// TIA Portal project "kanalAlarmowySygDzwiek" (V15)

(* hardware
DEVICE "S7-1200 station_1"  S7-1200 Station
   slot 0: "Rack_0"  S7-1200 Rack  Rack  V1.0
   slot 1: "PLC_1"  CPU 1214C DC/DC/DC  6ES7 214-1AG40-0XB0  V4.2
      slot 3: "AQ 1x12BIT_1"  AQ1 signal board  6ES7 232-4HA30-0XB0  V1.0
   slot 101: "CM 1243-5"  CM 1243-5  6GK7 243-5DX30-0XE0  V1.3
   slot 102: "CM 1241 (RS485)_1"  CM 1241 (RS485)  6ES7 241-1CH30-0XB0  V1.0
DEVICE "S7-1200 station_2"  S7-1200 Station
   slot 0: "Rack_0"  S7-1200 Rack  Rack  V1.0
   slot 1: "PLC_2"  CPU 1212C DC/DC/DC  6ES7 212-1AE40-0XB0  V4.2
   slot 2: "AI 4x13BIT/AQ 2x14BIT_1"  6ES7 234-4HE32-0XB0  V2.0
*)

// ===== PLC "PLC_1"  CPU 1214C DC/DC/DC =====

VAR_GLOBAL   // PLC tag table "Default tag table"
   "Clock_Byte" AT %MB50 : Byte;
   "Clock_10Hz" AT %M50.0 : Bool;
   "Clock_5Hz" AT %M50.1 : Bool;
   "Clock_2.5Hz" AT %M50.2 : Bool;
   "Clock_2Hz" AT %M50.3 : Bool;
   "Clock_1.25Hz" AT %M50.4 : Bool;
   "Clock_1Hz" AT %M50.5 : Bool;
   "Clock_0.625Hz" AT %M50.6 : Bool;
   "Clock_0.5Hz" AT %M50.7 : Bool;
   "System_Byte" AT %MB1 : Byte;
   "FirstScan" AT %M1.0 : Bool;
   "DiagStatusUpdate" AT %M1.1 : Bool;
   "AlwaysTRUE" AT %M1.2 : Bool;
   "AlwaysFALSE" AT %M1.3 : Bool;
   "zaklocenie" AT %I0.0 : Bool;
   "potwierdzenie" AT %I0.7 : Bool;
   "Tag_1" AT %M10.0 : Bool;
   "Tag_2" AT %M10.1 : Bool;
   "sygnalizacja" AT %Q0.1 : Bool;
   "System_Byte(1)" AT %MB1 : Byte;
   "Tag_3" AT %I0.1 : Bool;
   "Tag_4" AT %I0.6 : Bool;
   "Tag_5" AT %M20.0 : Bool;
   "Tag_6" AT %Q0.2 : Bool;
   "czasTrwania" AT %MD30 : Time;
   "Tag_7" AT %M22.0 : Bool;
   "Tag_8" AT %M22.1 : Bool;
   "Tag_9" AT %M22.2 : Bool;
   "Tag_10" AT %M22.3 : Bool;
   "Tag_11" AT %Q0.3 : Bool;
   "Tag_12" AT %I0.3 : Bool;
   "Tag_13" AT %I0.4 : Bool;
   "Tag_14" AT %I0.5 : Bool;
END_VAR

DATA_BLOCK "kanalAlarmowyFiltracja_DB"   // DB2
{ S7_Optimized_Access := 'TRUE' }
VERSION : 0.1
// stored: InstanceOfName kanalAlarmowyFiltracja
"kanalAlarmowyFiltracja"
BEGIN
END_DATA_BLOCK

DATA_BLOCK "kanalAlarmowyAnalogowy_DB"   // DB3
{ S7_Optimized_Access := 'TRUE' }
VERSION : 0.1
// stored: InstanceOfName kanalAlarmowyAnalogowy
"kanalAlarmowyAnalogowy"
BEGIN
END_DATA_BLOCK

// folder: System blocks/Program resources

DATA_BLOCK "IEC_Counter_0_DB"   // DB1
{ S7_Optimized_Access := 'TRUE' }
AUTHOR : Simatic
FAMILY : IEC
NAME : CNTR
VERSION : 1.0
// stored: InstanceOfName IEC_COUNTER
"IEC_COUNTER"
BEGIN
END_DATA_BLOCK

// folder: (top level)

FUNCTION_BLOCK "kanalAlarmowyFiltracja"   // FB1, LAD
{ S7_Optimized_Access := 'TRUE' }
VERSION : 0.1
   VAR_INPUT
      zaklocenie : Bool;
      potwierdzenie : Bool;
   END_VAR
   VAR_OUTPUT
      sygnalizacja : Bool;
   END_VAR
   VAR_IN_OUT
      pamAwarii : Bool;
      genSzpilki : Bool;
      czasTrwania : Time;
   END_VAR
   VAR
      IEC_Timer_0_Instance : TON_TIME;
   END_VAR
BEGIN

REGION Network 1
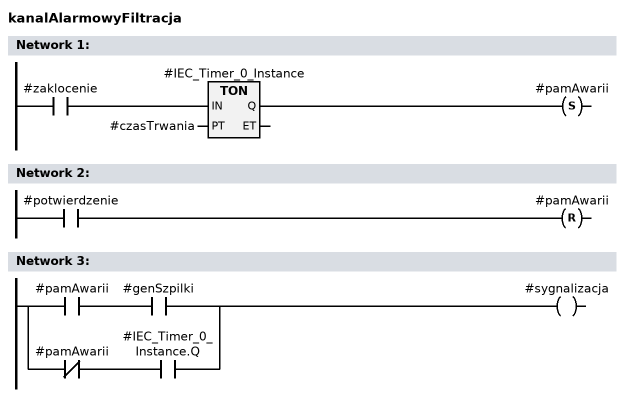
   #IEC_Timer_0_Instance(IN := #zaklocenie, PT := #czasTrwania);   // TON
   IF #IEC_Timer_0_Instance.Q THEN #pamAwarii := TRUE; END_IF;
END_REGION

REGION Network 2
   RUNG wire#powerrail
      Contact( #potwierdzenie )
      R_Coil( #pamAwarii )
   END_RUNG
   // the same network as SCL:
   IF #potwierdzenie THEN #pamAwarii := FALSE; END_IF;
END_REGION

REGION Network 3
   RUNG wire#powerrail
      Contact( #pamAwarii )
      Contact( #genSzpilki )
      wire#w1
      Coil( #sygnalizacja )
   END_RUNG
   RUNG wire#powerrail
      I_Contact( #pamAwarii )
      Contact( #IEC_Timer_0_Instance.Q )
   END_RUNG wire#w1
   // the same network as SCL:
   #sygnalizacja := (#pamAwarii AND #genSzpilki) OR (NOT #pamAwarii AND #IEC_Timer_0_Instance.Q);
END_REGION
END_FUNCTION_BLOCK

FUNCTION_BLOCK "kanalAlarmowyAnalogowy"   // FB2, LAD
{ S7_Optimized_Access := 'TRUE' }
VERSION : 0.1
   VAR_INPUT
      zaklocenie1 : Bool;
      pomiar2Analog : Int;
      granicaG : Int := 7;
      granicaD : Int := 2;
   END_VAR
   VAR_OUTPUT
      syngalizacja : Bool;
   END_VAR
   VAR_IN_OUT
      pamZaklocenia1 : Bool;
      pamZaklocenia2A : Bool;
      pamAwarii : Bool;
      pamZboczaZaklocenia2 : Bool;
      generatorSzpilki : Bool;
      potwierdzenie : Bool;
   END_VAR
   VAR_TEMP   // added for the SCL form of the ladder/FBD networks
      _w1 : Bool;
      _w2 : Bool;
   END_VAR
BEGIN

REGION Network 1: wykrycie awarii
   // 2 kanaly
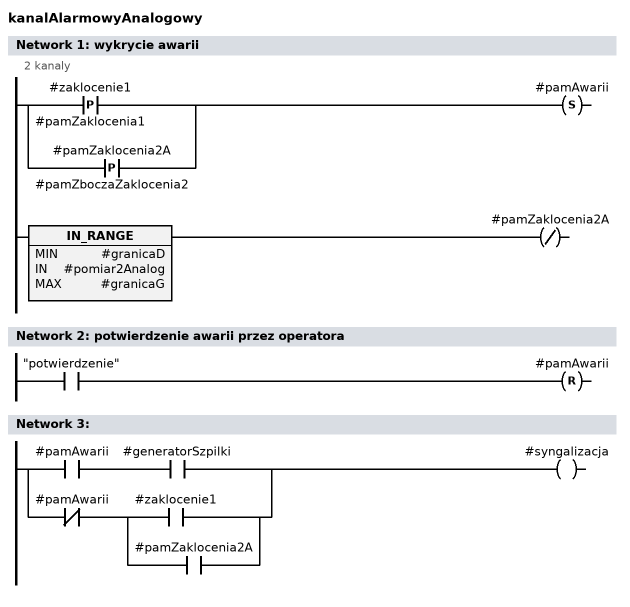
   RUNG wire#powerrail
      P_Contact(operand := #zaklocenie1, bit := #pamZaklocenia1)
      wire#w1
      S_Coil( #pamAwarii )
   END_RUNG
   RUNG wire#powerrail
      P_Contact(operand := #pamZaklocenia2A, bit := #pamZboczaZaklocenia2)
   END_RUNG wire#w1
   RUNG wire#powerrail
      { S7_Templates := "SrcType := Int" } InRange(min := #granicaD, in := #pomiar2Analog, max := #granicaG)
      I_Coil( #pamZaklocenia2A )
   END_RUNG
   // the same network as SCL:
   #_w1 := #zaklocenie1 AND NOT #pamZaklocenia1;   // rising edge of #zaklocenie1
   #pamZaklocenia1 := #zaklocenie1;
   #_w2 := #pamZaklocenia2A AND NOT #pamZboczaZaklocenia2;   // rising edge of #pamZaklocenia2A
   #pamZboczaZaklocenia2 := #pamZaklocenia2A;
   IF #_w1 OR #_w2 THEN #pamAwarii := TRUE; END_IF;
   #pamZaklocenia2A := NOT ((#granicaD <= #pomiar2Analog) AND (#pomiar2Analog <= #granicaG));
END_REGION

REGION Network 2: potwierdzenie awarii przez operatora
   RUNG wire#powerrail
      Contact( "potwierdzenie" )
      R_Coil( #pamAwarii )
   END_RUNG
   // the same network as SCL:
   IF "potwierdzenie" THEN #pamAwarii := FALSE; END_IF;
END_REGION

REGION Network 3
   RUNG wire#powerrail
      Contact( #pamAwarii )
      Contact( #generatorSzpilki )
      wire#w1
      Coil( #syngalizacja )
   END_RUNG
   RUNG wire#powerrail
      I_Contact( #pamAwarii )
      wire#w2
      Contact( #zaklocenie1 )
   END_RUNG wire#w1
   RUNG wire#w2
      Contact( #pamZaklocenia2A )
   END_RUNG wire#w1
   // the same network as SCL:
   #syngalizacja := (#pamAwarii AND #generatorSzpilki) OR (NOT #pamAwarii AND (#zaklocenie1 OR #pamZaklocenia2A));
END_REGION
END_FUNCTION_BLOCK

FUNCTION "kanalAlarmowy" : Void   // FC1, LAD
{ S7_Optimized_Access := 'TRUE' }
VERSION : 0.1
   VAR_INPUT
      zaklocenie : Bool;
      potwierdzenie : Bool;
   END_VAR
   VAR_OUTPUT
      sygnalizacja : Bool;
   END_VAR
   VAR_IN_OUT
      pamZbocza : Bool;
      pamAwarii : Bool;
      generatorSzpilki : Bool;
   END_VAR
   VAR_TEMP   // added for the SCL form of the ladder/FBD networks
      _w1 : Bool;
   END_VAR
BEGIN

REGION Network 1: Wykrycie zakłócenie awarii
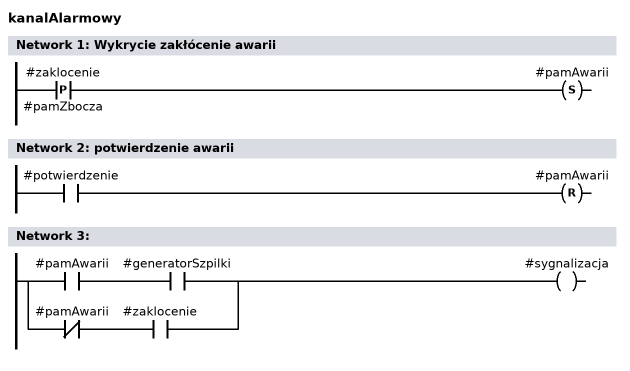
   RUNG wire#powerrail
      P_Contact(operand := #zaklocenie, bit := #pamZbocza)
      S_Coil( #pamAwarii )
   END_RUNG
   // the same network as SCL:
   #_w1 := #zaklocenie AND NOT #pamZbocza;   // rising edge of #zaklocenie
   #pamZbocza := #zaklocenie;
   IF #_w1 THEN #pamAwarii := TRUE; END_IF;
END_REGION

REGION Network 2: potwierdzenie awarii
   RUNG wire#powerrail
      Contact( #potwierdzenie )
      R_Coil( #pamAwarii )
   END_RUNG
   // the same network as SCL:
   IF #potwierdzenie THEN #pamAwarii := FALSE; END_IF;
END_REGION

REGION Network 3
   RUNG wire#powerrail
      Contact( #pamAwarii )
      Contact( #generatorSzpilki )
      wire#w1
      Coil( #sygnalizacja )
   END_RUNG
   RUNG wire#powerrail
      I_Contact( #pamAwarii )
      Contact( #zaklocenie )
   END_RUNG wire#w1
   // the same network as SCL:
   #sygnalizacja := (#pamAwarii AND #generatorSzpilki) OR (NOT #pamAwarii AND #zaklocenie);
END_REGION
END_FUNCTION

ORGANIZATION_BLOCK "Main"   // OB1, LAD, ProgramCycle
TITLE = "Main Program Sweep (Cycle)"
{ S7_Optimized_Access := 'TRUE' }
VERSION : 0.1
   VAR_INPUT
      Initial_Call : Bool;   // Initial call of this OB
      Remanence : Bool;   // =True, if remanent data are available
   END_VAR
BEGIN

REGION Network 1: zwykły kanał alarmowy FC
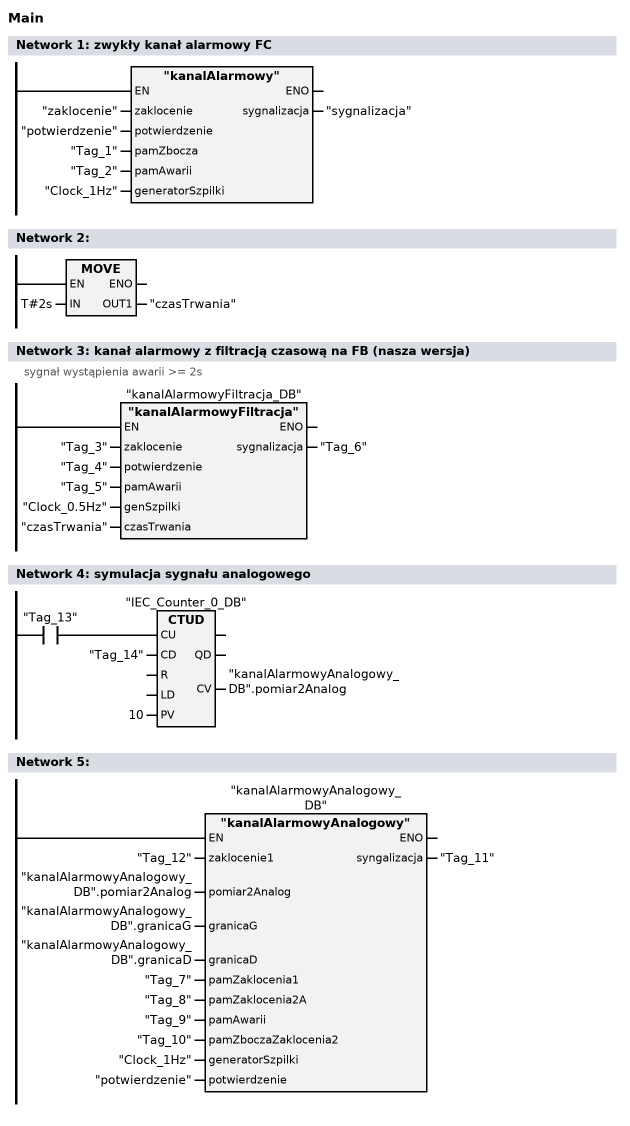
   RUNG wire#powerrail
      "kanalAlarmowy"(zaklocenie := "zaklocenie", potwierdzenie := "potwierdzenie", pamZbocza := "Tag_1", pamAwarii := "Tag_2", generatorSzpilki := "Clock_1Hz", sygnalizacja => "sygnalizacja")
   END_RUNG
   // the same network as SCL:
   "kanalAlarmowy"(zaklocenie := "zaklocenie",
                   potwierdzenie := "potwierdzenie",
                   pamZbocza := "Tag_1",
                   pamAwarii := "Tag_2",
                   generatorSzpilki := "Clock_1Hz",
                   sygnalizacja => "sygnalizacja");
END_REGION

REGION Network 2
   RUNG wire#powerrail
      Move(in := T#2s, out1 => "czasTrwania")
   END_RUNG
   // the same network as SCL:
   "czasTrwania" := T#2s;
END_REGION

REGION Network 3: kanał alarmowy z filtracją czasową na FB (nasza wersja)
   // sygnał wystąpienia awarii >= 2s
   RUNG wire#powerrail
      "kanalAlarmowyFiltracja_DB"(zaklocenie := "Tag_3", potwierdzenie := "Tag_4", pamAwarii := "Tag_5", genSzpilki := "Clock_0.5Hz", czasTrwania := "czasTrwania", sygnalizacja => "Tag_6")
   END_RUNG
   // the same network as SCL:
   "kanalAlarmowyFiltracja_DB"(zaklocenie := "Tag_3",   // "kanalAlarmowyFiltracja"
                           potwierdzenie := "Tag_4",
                           pamAwarii := "Tag_5",
                           genSzpilki := "Clock_0.5Hz",
                           czasTrwania := "czasTrwania",
                           sygnalizacja => "Tag_6");
END_REGION

REGION Network 4: symulacja sygnału analogowego
   "IEC_Counter_0_DB".CTUD(CU := "Tag_13",
                           CD := "Tag_14",
                           PV := 10,
                           CV => "kanalAlarmowyAnalogowy_DB".pomiar2Analog);
END_REGION

REGION Network 5
   RUNG wire#powerrail
      "kanalAlarmowyAnalogowy_DB"(zaklocenie1 := "Tag_12", pomiar2Analog := "kanalAlarmowyAnalogowy_DB".pomiar2Analog, granicaG := "kanalAlarmowyAnalogowy_DB".granicaG, granicaD := "kanalAlarmowyAnalogowy_DB".granicaD, pamZaklocenia1 := "Tag_7", pamZaklocenia2A := "Tag_8", pamAwarii := "Tag_9", pamZboczaZaklocenia2 := "Tag_10", generatorSzpilki := "Clock_1Hz", potwierdzenie := "potwierdzenie", syngalizacja => "Tag_11")
   END_RUNG
   // the same network as SCL:
   "kanalAlarmowyAnalogowy_DB"(zaklocenie1 := "Tag_12",   // "kanalAlarmowyAnalogowy"
                           pomiar2Analog := "kanalAlarmowyAnalogowy_DB".pomiar2Analog,
                           granicaG := "kanalAlarmowyAnalogowy_DB".granicaG,
                           granicaD := "kanalAlarmowyAnalogowy_DB".granicaD,
                           pamZaklocenia1 := "Tag_7",
                           pamZaklocenia2A := "Tag_8",
                           pamAwarii := "Tag_9",
                           pamZboczaZaklocenia2 := "Tag_10",
                           generatorSzpilki := "Clock_1Hz",
                           potwierdzenie := "potwierdzenie",
                           syngalizacja => "Tag_11");
END_REGION
END_ORGANIZATION_BLOCK

// ===== PLC "PLC_2"  CPU 1212C DC/DC/DC =====

VAR_GLOBAL   // PLC tag table "Default tag table"
   "Tag_15" AT %I0.0 : Bool;
   "Tag_16" AT %I0.7 : Bool;
   "Tag_1" AT %M10.0 : Bool;
   "Tag_17" AT %M10.1 : Bool;
   "Tag_18" AT %Q0.0 : Bool;
   "Clock_Byte" AT %MB50 : Byte;
   "Clock_10Hz" AT %M50.0 : Bool;
   "Clock_5Hz" AT %M50.1 : Bool;
   "Clock_2.5Hz" AT %M50.2 : Bool;
   "Clock_2Hz" AT %M50.3 : Bool;
   "Clock_1.25Hz" AT %M50.4 : Bool;
   "Clock_1Hz" AT %M50.5 : Bool;
   "Clock_0.625Hz" AT %M50.6 : Bool;
   "Clock_0.5Hz" AT %M50.7 : Bool;
   "Tag_19" AT %I0.2 : Bool;
   "Tag_20" AT %I0.6 : Bool;
   "Tag_21" AT %M20.2 : Bool;
   "Tag_22" AT %M20.3 : Bool;
   "Tag_23" AT %Q0.1 : Bool;
   "Tag_24" AT %I0.3 : Bool;
   "Tag_25" AT %I0.4 : Bool;
   "Tag_26" AT %I0.5 : Bool;
   "Tag_27" AT %Q0.3 : Bool;
   "Tag_28" AT %M24.0 : Bool;
   "Tag_29" AT %M24.1 : Bool;
   "Tag_30" AT %M24.2 : Bool;
   "Tag_31" AT %M24.3 : Bool;
   "czasTrwania" AT %MD32 : Time;
END_VAR

DATA_BLOCK "kanalAlarmowyFiltracja_DB"   // DB2
{ S7_Optimized_Access := 'TRUE' }
VERSION : 0.1
// stored: InstanceOfName kanalAlarmowyFiltracja
"kanalAlarmowyFiltracja"
BEGIN
END_DATA_BLOCK

DATA_BLOCK "kanalAlarmowyAnalogowy_DB"   // DB3
{ S7_Optimized_Access := 'TRUE' }
VERSION : 0.1
// stored: InstanceOfName kanalAlarmowyAnalogowy
"kanalAlarmowyAnalogowy"
BEGIN
END_DATA_BLOCK

// folder: System blocks/Program resources

DATA_BLOCK "IEC_Counter_0_DB"   // DB1
{ S7_Optimized_Access := 'TRUE' }
AUTHOR : Simatic
FAMILY : IEC
NAME : CNTR
VERSION : 1.0
// stored: InstanceOfName IEC_COUNTER
"IEC_COUNTER"
BEGIN
END_DATA_BLOCK

// folder: (top level)

FUNCTION_BLOCK "kanalAlarmowyFiltracja"   // FB1, LAD
{ S7_Optimized_Access := 'TRUE' }
VERSION : 0.1
   VAR_INPUT
      zaklocenie : Bool;
      potwierdzenie : Bool;
   END_VAR
   VAR_OUTPUT
      sygnalizacja : Bool;
   END_VAR
   VAR_IN_OUT
      pamAwarii : Bool;
      genSzpilki : Bool;
      czasTrwania : Time;
   END_VAR
   VAR
      IEC_Timer_0_Instance : TON_TIME;
   END_VAR
BEGIN

REGION Network 1
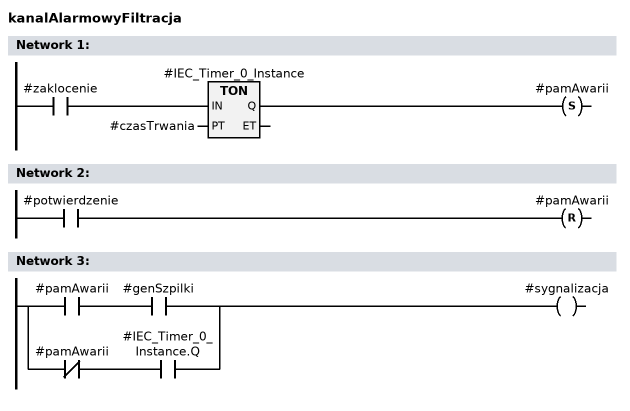
   #IEC_Timer_0_Instance(IN := #zaklocenie, PT := #czasTrwania);   // TON
   IF #IEC_Timer_0_Instance.Q THEN #pamAwarii := TRUE; END_IF;
END_REGION

REGION Network 2
   RUNG wire#powerrail
      Contact( #potwierdzenie )
      R_Coil( #pamAwarii )
   END_RUNG
   // the same network as SCL:
   IF #potwierdzenie THEN #pamAwarii := FALSE; END_IF;
END_REGION

REGION Network 3
   RUNG wire#powerrail
      Contact( #pamAwarii )
      Contact( #genSzpilki )
      wire#w1
      Coil( #sygnalizacja )
   END_RUNG
   RUNG wire#powerrail
      I_Contact( #pamAwarii )
      Contact( #IEC_Timer_0_Instance.Q )
   END_RUNG wire#w1
   // the same network as SCL:
   #sygnalizacja := (#pamAwarii AND #genSzpilki) OR (NOT #pamAwarii AND #IEC_Timer_0_Instance.Q);
END_REGION
END_FUNCTION_BLOCK

FUNCTION_BLOCK "kanalAlarmowyAnalogowy"   // FB2, LAD
{ S7_Optimized_Access := 'TRUE' }
VERSION : 0.1
   VAR_INPUT
      zaklocenie1 : Bool;
      pomiar2Analog : Int;
      granicaG : Int := 7;
      granicaD : Int := 2;
   END_VAR
   VAR_OUTPUT
      syngalizacja : Bool;
   END_VAR
   VAR_IN_OUT
      pamZaklocenia1 : Bool;
      pamZaklocenia2A : Bool;
      pamAwarii : Bool;
      pamZboczaZaklocenia2 : Bool;
      generatorSzpilki : Bool;
      potwierdzenie : Bool;
   END_VAR
   VAR_TEMP   // added for the SCL form of the ladder/FBD networks
      _w1 : Bool;
      _w2 : Bool;
   END_VAR
BEGIN

REGION Network 1: wykrycie awarii
   // 2 kanaly
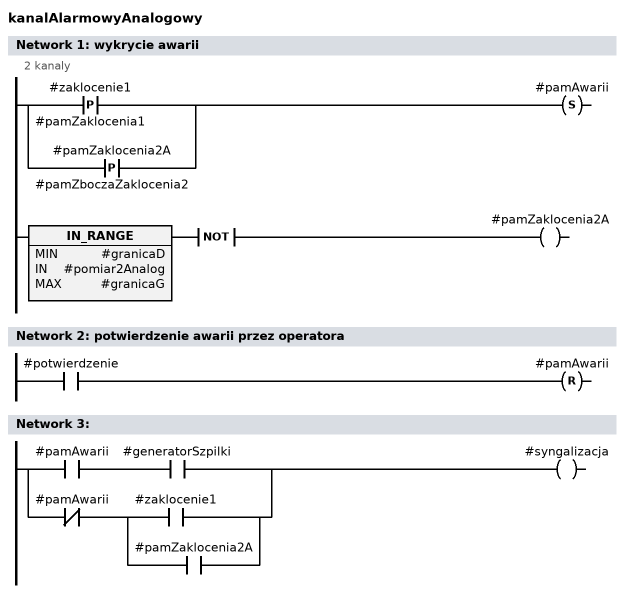
   RUNG wire#powerrail
      P_Contact(operand := #zaklocenie1, bit := #pamZaklocenia1)
      wire#w1
      S_Coil( #pamAwarii )
   END_RUNG
   RUNG wire#powerrail
      P_Contact(operand := #pamZaklocenia2A, bit := #pamZboczaZaklocenia2)
   END_RUNG wire#w1
   RUNG wire#powerrail
      { S7_Templates := "SrcType := Int" } InRange(min := #granicaD, in := #pomiar2Analog, max := #granicaG)
      Not()
      Coil( #pamZaklocenia2A )
   END_RUNG
   // the same network as SCL:
   #_w1 := #zaklocenie1 AND NOT #pamZaklocenia1;   // rising edge of #zaklocenie1
   #pamZaklocenia1 := #zaklocenie1;
   #_w2 := #pamZaklocenia2A AND NOT #pamZboczaZaklocenia2;   // rising edge of #pamZaklocenia2A
   #pamZboczaZaklocenia2 := #pamZaklocenia2A;
   IF #_w1 OR #_w2 THEN #pamAwarii := TRUE; END_IF;
   #pamZaklocenia2A := NOT ((#granicaD <= #pomiar2Analog) AND (#pomiar2Analog <= #granicaG));
END_REGION

REGION Network 2: potwierdzenie awarii przez operatora
   RUNG wire#powerrail
      Contact( #potwierdzenie )
      R_Coil( #pamAwarii )
   END_RUNG
   // the same network as SCL:
   IF #potwierdzenie THEN #pamAwarii := FALSE; END_IF;
END_REGION

REGION Network 3
   RUNG wire#powerrail
      Contact( #pamAwarii )
      Contact( #generatorSzpilki )
      wire#w1
      Coil( #syngalizacja )
   END_RUNG
   RUNG wire#powerrail
      I_Contact( #pamAwarii )
      wire#w2
      Contact( #zaklocenie1 )
   END_RUNG wire#w1
   RUNG wire#w2
      Contact( #pamZaklocenia2A )
   END_RUNG wire#w1
   // the same network as SCL:
   #syngalizacja := (#pamAwarii AND #generatorSzpilki) OR (NOT #pamAwarii AND (#zaklocenie1 OR #pamZaklocenia2A));
END_REGION
END_FUNCTION_BLOCK

FUNCTION "kanalAlarmowy" : Void   // FC1, LAD
{ S7_Optimized_Access := 'TRUE' }
VERSION : 0.1
   VAR_INPUT
      zaklocenie : Bool;
      potwierdzenie : Bool;
   END_VAR
   VAR_OUTPUT
      sygnalizacja : Bool;
   END_VAR
   VAR_IN_OUT
      pamZbocza : Bool;
      pamAwarii : Bool;
      generatorSzpilki : Bool;
   END_VAR
   VAR_TEMP   // added for the SCL form of the ladder/FBD networks
      _w1 : Bool;
   END_VAR
BEGIN

REGION Network 1: Wykrycie zakłócenie awarii
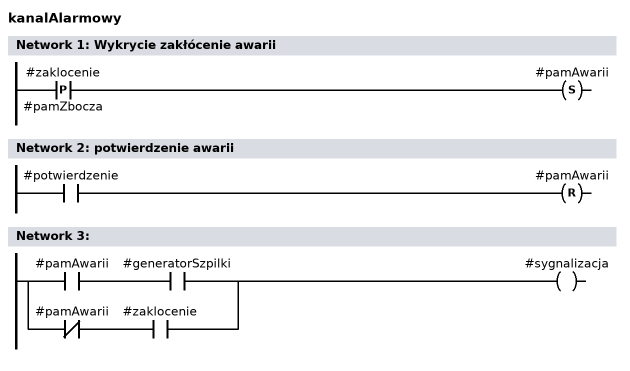
   RUNG wire#powerrail
      P_Contact(operand := #zaklocenie, bit := #pamZbocza)
      S_Coil( #pamAwarii )
   END_RUNG
   // the same network as SCL:
   #_w1 := #zaklocenie AND NOT #pamZbocza;   // rising edge of #zaklocenie
   #pamZbocza := #zaklocenie;
   IF #_w1 THEN #pamAwarii := TRUE; END_IF;
END_REGION

REGION Network 2: potwierdzenie awarii
   RUNG wire#powerrail
      Contact( #potwierdzenie )
      R_Coil( #pamAwarii )
   END_RUNG
   // the same network as SCL:
   IF #potwierdzenie THEN #pamAwarii := FALSE; END_IF;
END_REGION

REGION Network 3
   RUNG wire#powerrail
      Contact( #pamAwarii )
      Contact( #generatorSzpilki )
      wire#w1
      Coil( #sygnalizacja )
   END_RUNG
   RUNG wire#powerrail
      I_Contact( #pamAwarii )
      Contact( #zaklocenie )
   END_RUNG wire#w1
   // the same network as SCL:
   #sygnalizacja := (#pamAwarii AND #generatorSzpilki) OR (NOT #pamAwarii AND #zaklocenie);
END_REGION
END_FUNCTION

ORGANIZATION_BLOCK "Main"   // OB1, LAD, ProgramCycle
TITLE = "Main Program Sweep (Cycle)"
{ S7_Optimized_Access := 'TRUE' }
VERSION : 0.1
   VAR_INPUT
      Initial_Call : Bool;   // Initial call of this OB
      Remanence : Bool;   // =True, if remanent data are available
   END_VAR
BEGIN

REGION Network 1: zwykły kanał alarmowy FC
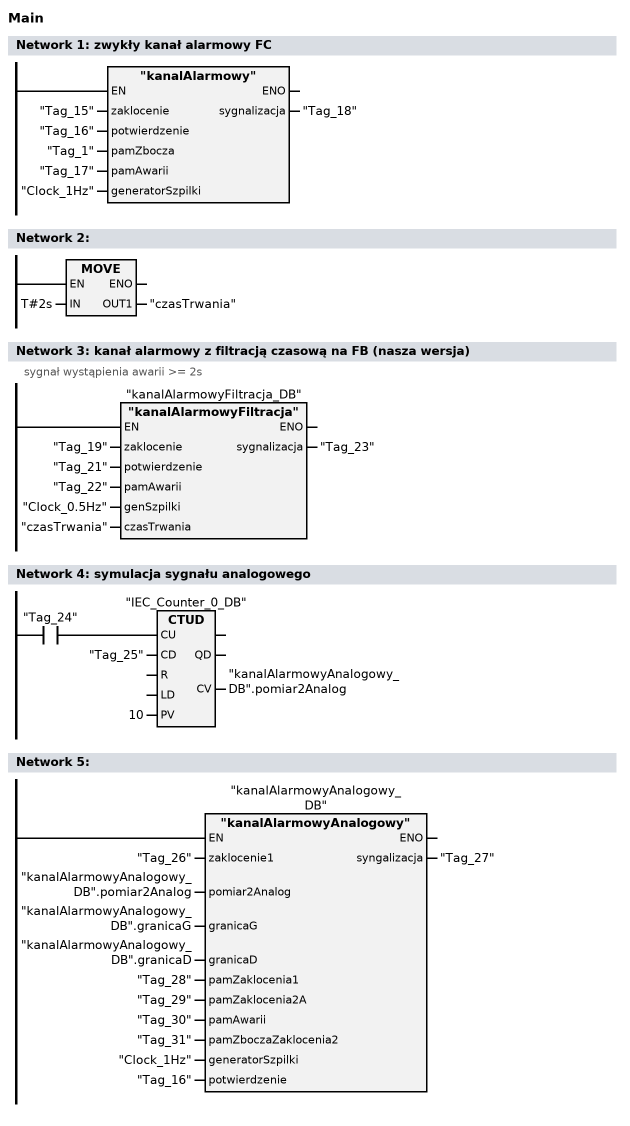
   RUNG wire#powerrail
      "kanalAlarmowy"(zaklocenie := "Tag_15", potwierdzenie := "Tag_16", pamZbocza := "Tag_1", pamAwarii := "Tag_17", generatorSzpilki := "Clock_1Hz", sygnalizacja => "Tag_18")
   END_RUNG
   // the same network as SCL:
   "kanalAlarmowy"(zaklocenie := "Tag_15",
                   potwierdzenie := "Tag_16",
                   pamZbocza := "Tag_1",
                   pamAwarii := "Tag_17",
                   generatorSzpilki := "Clock_1Hz",
                   sygnalizacja => "Tag_18");
END_REGION

REGION Network 2
   RUNG wire#powerrail
      Move(in := T#2s, out1 => "czasTrwania")
   END_RUNG
   // the same network as SCL:
   "czasTrwania" := T#2s;
END_REGION

REGION Network 3: kanał alarmowy z filtracją czasową na FB (nasza wersja)
   // sygnał wystąpienia awarii >= 2s
   RUNG wire#powerrail
      "kanalAlarmowyFiltracja_DB"(zaklocenie := "Tag_19", potwierdzenie := "Tag_21", pamAwarii := "Tag_22", genSzpilki := "Clock_0.5Hz", czasTrwania := "czasTrwania", sygnalizacja => "Tag_23")
   END_RUNG
   // the same network as SCL:
   "kanalAlarmowyFiltracja_DB"(zaklocenie := "Tag_19",   // "kanalAlarmowyFiltracja"
                           potwierdzenie := "Tag_21",
                           pamAwarii := "Tag_22",
                           genSzpilki := "Clock_0.5Hz",
                           czasTrwania := "czasTrwania",
                           sygnalizacja => "Tag_23");
END_REGION

REGION Network 4: symulacja sygnału analogowego
   "IEC_Counter_0_DB".CTUD(CU := "Tag_24",
                           CD := "Tag_25",
                           PV := 10,
                           CV => "kanalAlarmowyAnalogowy_DB".pomiar2Analog);
END_REGION

REGION Network 5
   RUNG wire#powerrail
      "kanalAlarmowyAnalogowy_DB"(zaklocenie1 := "Tag_26", pomiar2Analog := "kanalAlarmowyAnalogowy_DB".pomiar2Analog, granicaG := "kanalAlarmowyAnalogowy_DB".granicaG, granicaD := "kanalAlarmowyAnalogowy_DB".granicaD, pamZaklocenia1 := "Tag_28", pamZaklocenia2A := "Tag_29", pamAwarii := "Tag_30", pamZboczaZaklocenia2 := "Tag_31", generatorSzpilki := "Clock_1Hz", potwierdzenie := "Tag_16", syngalizacja => "Tag_27")
   END_RUNG
   // the same network as SCL:
   "kanalAlarmowyAnalogowy_DB"(zaklocenie1 := "Tag_26",   // "kanalAlarmowyAnalogowy"
                           pomiar2Analog := "kanalAlarmowyAnalogowy_DB".pomiar2Analog,
                           granicaG := "kanalAlarmowyAnalogowy_DB".granicaG,
                           granicaD := "kanalAlarmowyAnalogowy_DB".granicaD,
                           pamZaklocenia1 := "Tag_28",
                           pamZaklocenia2A := "Tag_29",
                           pamAwarii := "Tag_30",
                           pamZboczaZaklocenia2 := "Tag_31",
                           generatorSzpilki := "Clock_1Hz",
                           potwierdzenie := "Tag_16",
                           syngalizacja => "Tag_27");
END_REGION
END_ORGANIZATION_BLOCK